{attribute addProperty BoxType "EL6002-0000-0019"}
{attribute addProperty Id "AdsAddrAT %I*AMSADDR6480StateAT %I*UINT1620"}
{attribute addProperty CRC "3160658815"}
{attribute addProperty SizeInBites "80"}
{attribute addProperty SizeInBytes "10"}
TYPE InfoData_BC63D37F :
STRUCT
	{attribute addProperty Name "AdsAddr"}
	AdsAddr AT %I* : AMSADDR;
	{attribute addProperty Name "State"}
	State AT %I* : UINT;
END_STRUCT
END_TYPE

(* stored: Version 1.2.0.0, ProductVersion 3.1.4024.9
   DUT InfoData_BC63D37F: Id {34a02ef5-23d4-07b7-15ca-957ff922c2f2} *)
